FUNCTION_BLOCK FB_Actor
VAR_INPUT
END_VAR
VAR_OUTPUT
END_VAR
VAR
	Actor AT %Q*:BOOL;
END_VAR

METHOD isActive : BOOL
VAR_INPUT
END_VAR
isActive:=Actor;
END_METHOD

METHOD setState : BOOL
VAR_INPUT
	input_state:bool;
END_VAR
Actor:=input_state;
END_METHOD

METHOD Start : BOOL
VAR_INPUT
END_VAR
Actor:=true;
END_METHOD

METHOD Stop : BOOL
VAR_INPUT
END_VAR
Actor:=false;
END_METHOD

METHOD Toggle : BOOL
VAR_INPUT
END_VAR
Actor:=not Actor;
END_METHOD

END_FUNCTION_BLOCK

(* stored: Version 1.1.0.1, ProductVersion 3.1.4022.9
   POU FB_Actor: Id {a6cdb25e-faff-4ea9-8b03-4bb80a8c6fec}, SpecialFunc None
   Method isActive: Id {ee71c033-2365-40f7-b2cf-06fe6b1de09c}
   Method setState: Id {f4de77f2-8abe-4e31-8885-38172aa43e1d}
   Method Start: Id {f2fc61c6-5da3-4394-bec3-39ce668b21e5}
   Method Stop: Id {2b8e146a-47f0-47a0-ab0f-de9cc3bb8113}
   Method Toggle: Id {be65ed87-3e59-47e8-97ed-779c0b5b83fa} *)
